// TIA Portal V19 export
DATA_BLOCK "Deckel_CM01"   // DB1190
// stored: AutoNumber false, InstanceOfName Deckel, InstanceOfType FB
"Deckel"
   // VAR
   //    In { ExternalAccessible := 'False'; ExternalVisible := 'False'; ExternalWritable := 'False'} : Struct
   //       NotHalt : Bool;
   //       Si_24VDC_links : Bool;
   //       Si_24VDC_rechts : Bool;
   //       Auto : Bool;
   //       Hand : Bool;
   //       Tipp : Bool;
   //       ErrQ : Bool;
   //       T_links_auf : Bool;
   //       T_links_zu : Bool;
   //       T_rechts_auf : Bool;
   //       T_rechts_zu : Bool;
   //       SRM_links_auf : Bool;
   //       SRM_links_zu : Bool;
   //       SRM_rechts_auf : Bool;
   //       SRM_rechts_zu : Bool;
   //       S_links_auf : Bool;
   //       S_links_zu : Bool;
   //       S_rechts_auf : Bool;
   //       S_rechts_zu : Bool;
   //    END_STRUCT;
   // END_VAR
   // VAR RETAIN
   //    Param { ExternalAccessible := 'False'; ExternalVisible := 'False'; ExternalWritable := 'False'} : Struct
   //       "TO" : Time;
   //       gleichzeitig : Time;
   //    END_STRUCT;
   //    Zst { ExternalAccessible := 'False'; ExternalVisible := 'False'; ExternalWritable := 'False'} : Struct
   //       Fehler : Bool;
   //       Sperre_Pos_li : Bool;
   //       Sperre_Pos_re : Bool;
   //       Req_links_auf : Bool;
   //       Req_rechts_auf : Bool;
   //       TW_sicher : Bool;
   //       Ist_Pos_links : Int;
   //       Ist_Pos_rechts : Int;
   //    END_STRUCT;
   //    Out { ExternalAccessible := 'False'; ExternalVisible := 'False'; ExternalWritable := 'False'} : Struct
   //       links_auf : Bool;
   //       links_zu : Bool;
   //       rechts_auf : Bool;
   //       rechts_zu : Bool;
   //    END_STRUCT;
   //    Mld { ExternalAccessible := 'False'; ExternalVisible := 'False'; ExternalWritable := 'False'} : Struct
   //       TO_links_auf : Bool;
   //       TO_links_zu : Bool;
   //       TO_rechts_auf : Bool;
   //       TO_rechts_zu : Bool;
   //       Si_24VDC_links : Bool;
   //       Si_24VDC_rechts : Bool;
   //       n_Auto : Bool;
   //       SF_gleich_li_auf : Bool;
   //       SF_gleich_li_zu : Bool;
   //       SF_gleich_re_auf : Bool;
   //       SF_gleich_re_zu : Bool;
   //    END_STRUCT;
   // END_VAR
   // VAR
   //    IEC_Timer { ExternalAccessible := 'False'; ExternalVisible := 'False'; ExternalWritable := 'False'} : Struct
   //       TO_li_auf { S7_SetPoint := 'True'} : TON_TIME;
   //       TO_li_zu { S7_SetPoint := 'True'} : TON_TIME;
   //       TO_re_auf { S7_SetPoint := 'True'} : TON_TIME;
   //       TO_re_zu { S7_SetPoint := 'True'} : TON_TIME;
   //       gleich_li_auf { S7_SetPoint := 'True'} : TON_TIME;
   //       gleich_li_zu { S7_SetPoint := 'True'} : TON_TIME;
   //       gleich_re_auf { S7_SetPoint := 'True'} : TON_TIME;
   //       gleich_re_zu { S7_SetPoint := 'True'} : TON_TIME;
   //    END_STRUCT;
   // END_VAR
BEGIN
END_DATA_BLOCK
